// TwinCAT 3 PLC project PLC
// ProgramVersion: 3.1.4024.0
// libraries:
//   Tc2_Standard, * (Beckhoff Automation GmbH)
//   Tc2_System, * (Beckhoff Automation GmbH)
//   Tc3_Module, * (Beckhoff Automation GmbH)
// project tree:
//   / PlcTask.TcTTO
//   POUs/ MAIN.TcPOU, PumpControl01.TcPOU, PumpControl03.TcPOU, PumpControl02.TcPOU
//   POUs/Simulation/ Simulation.TcPOU
// real-time tasks:
//   TASK PlcTask: cycle T#10ms, priority 20, ADS port 350

CONFIGURATION PLC
    RESOURCE PLC ON TwinCAT3
        TASK PlcTask(INTERVAL := T#10ms, PRIORITY := 20);
        PROGRAM MAIN WITH PlcTask : MAIN;
    END_RESOURCE
END_CONFIGURATION

// ---- POUs/MAIN.TcPOU
PROGRAM MAIN
VAR
	PumpControl01				:	PumpControl01;
	PumpControl02				:	PumpControl02;
	PumpControl03				:	PumpControl03;
	M1_01: BOOL;
	M2_01: BOOL;
	M1_02: BOOL;
	M2_02: BOOL;
	M1_03: BOOL;
	M2_03: BOOL;
END_VAR

Simulation();
PumpControl01(LsLow := Simulation.LsLow, LsMiddle := Simulation.LsMiddle, LsHigh := Simulation.LsHigh);
M1_01 := PumpControl01.Motor1;
M2_01 := PumpControl01.Motor2;
PumpControl02(LsLow := Simulation.LsLow, LsMiddle := Simulation.LsMiddle, LsHigh := Simulation.LsHigh);
M1_02 := PumpControl02.Motor1;
M2_02 := PumpControl02.Motor2;
PumpControl02(LsLow := Simulation.LsLow, LsMiddle := Simulation.LsMiddle, LsHigh := Simulation.LsHigh);
M1_03 := PumpControl02.Motor1;
M2_03 := PumpControl02.Motor2;

END_PROGRAM

// ---- POUs/PumpControl01.TcPOU
FUNCTION_BLOCK PumpControl01
VAR_INPUT
	LsLow							:	BOOL;		// limit switch LOW (NO)
	LsMiddle						:	BOOL;		// limit switch MIDDLE (NO)
	LsHigh							:	BOOL;		// limit switch HIGH (NC)
END_VAR
VAR_OUTPUT
	Motor1							:	BOOL;		// motor 1 output
	Motor2							:	BOOL;		// motor 2 output
END_VAR
VAR
	AlternatePump					:	BOOL;		// flag for pump alternation
	RunMotor						:	BOOL;		// pump alternation control
END_VAR
VAR // added by the converter: edge detectors and wires of the graphical bodies
    _w1, _w2, _w3 : BOOL;
END_VAR

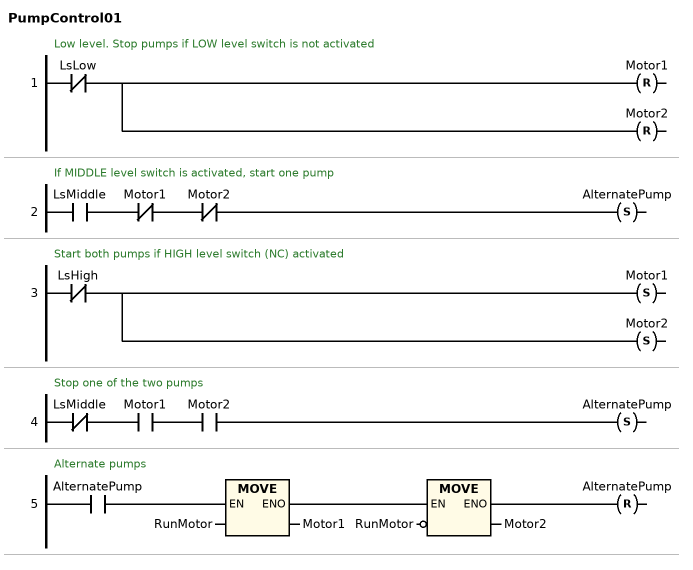
// NETWORK 1
// Low level. Stop pumps if LOW level switch is not activated
_w1 := NOT LsLow;
Motor1 R= _w1;
Motor2 R= _w1;

// NETWORK 2
// If MIDDLE level switch is activated, start one pump
AlternatePump S= LsMiddle AND NOT Motor1 AND NOT Motor2;

// NETWORK 3
// Start both pumps if HIGH level switch (NC) activated
_w2 := NOT LsHigh;
Motor1 S= _w2;
Motor2 S= _w2;

// NETWORK 4
// Stop one of the two pumps
AlternatePump S= NOT LsMiddle AND Motor1 AND Motor2;

// NETWORK 5
// Alternate pumps
_w3 := AlternatePump;
IF _w3 THEN Motor1 := RunMotor; END_IF
IF _w3 THEN Motor2 := NOT RunMotor; END_IF
AlternatePump R= _w3;

END_FUNCTION_BLOCK

// ---- POUs/PumpControl02.TcPOU
FUNCTION_BLOCK PumpControl02
VAR_INPUT
	LsLow							:	BOOL;		// limit switch LOW (NO)
	LsMiddle						:	BOOL;		// limit switch MIDDLE (NO)
	LsHigh							:	BOOL;		// limit switch HIGH (NC)
END_VAR
VAR_OUTPUT
	Motor1							:	BOOL;		// motor 1 output
	Motor2							:	BOOL;		// motor 2 output
END_VAR
VAR
	SeqStep							:	(INIT, LOW, MIDDLE, HIGH) := INIT;
	RunMotor						:	BOOL;		// pump alternation control
END_VAR

SeqSelect();
SeqOutput();

METHOD SeqOutput : BOOL
VAR_INPUT
END_VAR

VAR
	StepMiddleOneShot: R_TRIG;
END_VAR
VAR_INST // added by the converter: edge detectors and wires of the graphical bodies
    _w1, _w2, _w3 : BOOL;
END_VAR
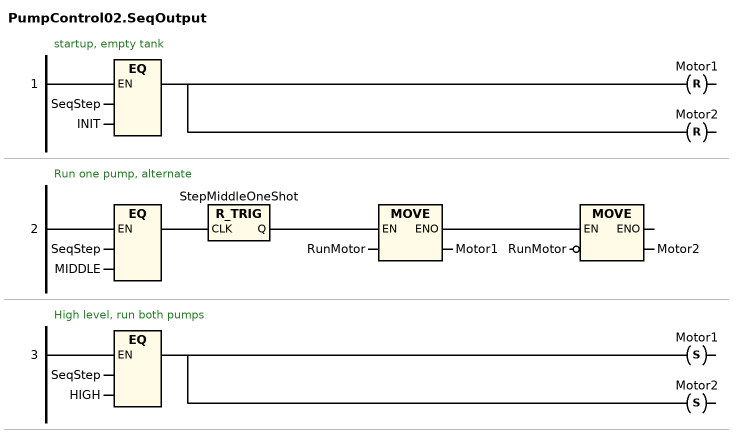
// NETWORK 1
// startup, empty tank
_w1 := SeqStep = INIT;
Motor1 R= _w1;
Motor2 R= _w1;

// NETWORK 2
// Run one pump, alternate
StepMiddleOneShot(CLK := SeqStep = MIDDLE); // R_TRIG
_w2 := StepMiddleOneShot.Q;
IF _w2 THEN Motor1 := RunMotor; END_IF
IF _w2 THEN Motor2 := NOT RunMotor; END_IF

// NETWORK 3
// High level, run both pumps
_w3 := SeqStep = HIGH;
Motor1 S= _w3;
Motor2 S= _w3;
END_METHOD

METHOD SeqSelect : BOOL
VAR_INPUT
END_VAR
VAR_INST // added by the converter: edge detectors and wires of the graphical bodies
    _w1 : BOOL;
END_VAR
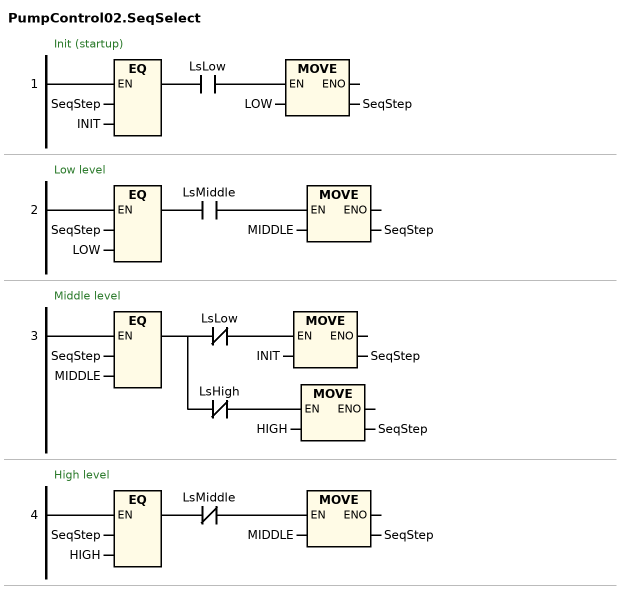
// NETWORK 1
// Init (startup)
IF SeqStep = INIT AND LsLow THEN SeqStep := LOW; END_IF

// NETWORK 2
// Low level
IF SeqStep = LOW AND LsMiddle THEN SeqStep := MIDDLE; END_IF

// NETWORK 3
// Middle level
_w1 := SeqStep = MIDDLE;
IF _w1 AND NOT LsLow THEN SeqStep := INIT; END_IF
IF _w1 AND NOT LsHigh THEN SeqStep := HIGH; END_IF

// NETWORK 4
// High level
IF SeqStep = HIGH AND NOT LsMiddle THEN SeqStep := MIDDLE; END_IF
END_METHOD

END_FUNCTION_BLOCK

// ---- POUs/PumpControl03.TcPOU
FUNCTION_BLOCK PumpControl03
VAR_INPUT
	LsLow							:	BOOL;		// limit switch LOW (NO)
	LsMiddle						:	BOOL;		// limit switch MIDDLE (NO)
	LsHigh							:	BOOL;		// limit switch HIGH (NC)
END_VAR
VAR_OUTPUT
	Motor1							:	BOOL;		// motor 1 output
	Motor2							:	BOOL;		// motor 2 output
END_VAR
VAR
	SeqStep							:	(STDBY, LOW, MIDDLE, HIGH) := STDBY;
	SeqStepOld						:	(STDBY, LOW, MIDDLE, HIGH);
	RunMotor						:	BOOL;		// pump alternation control
END_VAR

SeqSelect();
SeqOutput();

METHOD SeqOutput : BOOL
VAR_INPUT
END_VAR
CASE SeqStep OF
	LOW:				// pumps off
		Motor1 := FALSE;
		Motor2 := FALSE;
		
	MIDDLE:				// run one pump
		// alternate between pumps
		// change pump is first time run
		IF SeqStep <> SeqStepOld THEN
			RunMotor := NOT RunMotor;
		END_IF
		
		// turn pumps on or off
		Motor1 := RunMotor;
		Motor2 := NOT RunMotor;
	HIGH:				// tank full
		Motor1 := TRUE;
		Motor2 := TRUE;
END_CASE
END_METHOD

METHOD SeqSelect : BOOL
VAR_INPUT
END_VAR
// save current sequence step to handle alternation between pumps
SeqStepOld := SeqStep;

CASE SeqStep OF
	STDBY:						// standby, no liquid in tank
		IF LsLow THEN			// low level reached
			SeqStep := LOW;
		END_IF
		
	LOW:
		IF LsMiddle THEN		// middle level reached
			SeqStep := MIDDLE;
		END_IF
		
	MIDDLE:						// tank half full
		IF NOT LsLow THEN		// level -> lower
			SeqStep := LOW;
		END_IF
		
		IF NOT LsHigh THEN		// level -> higher
			SeqStep := HIGH;
		END_IF
	
	HIGH:						// tank full
		IF NOT LsMiddle THEN	// level -> lower
			SeqStep := MIDDLE;
		END_IF
END_CASE
END_METHOD

END_FUNCTION_BLOCK

// ---- POUs/Simulation/Simulation.TcPOU
PROGRAM Simulation
VAR
	Idx					:	REAL;
	Level				: 	REAL;
END_VAR

VAR_OUTPUT
	LsLow: BOOL;
	LsMiddle: BOOL;
	LsHigh: BOOL;
END_VAR

Idx := Idx + 0.001;
Level := SIN(Idx);

Level := Level * 2000 + 2000;

LsLow 		:= Level >= 1500;
LsMiddle 	:= Level >= 2500;
LsHigh		:= NOT (Level >= 3500);

END_PROGRAM
